// TIA Portal V19 export
FUNCTION "APP_UPDATE STEP NO. UHT" : Void   // FC30, STL
TITLE = Step update to OP25
{ S7_Optimized_Access := 'TRUE' }
AUTHOR : JOM
FAMILY : APP
NAME : STEP_UPD
// Main Update:       1 = Start                     7 = Stop production     
//                    2 = Presterilizing            8 = Recirculation water
//                    3 = Stop presteril            9 = Stop recirculation water
//                    4 = Cip                      10 = Aseptic cip
//                    5 = Stop cip                 11 = Stop aseptic cip
//                    6 = Production               12 = Total stop
//                    13 = CIP FILLER
// 
// Step Update:     101 = Standby             102-110 = Start     
//              111-120 = Presterilizing      121-130 = Stop presteril
//              131-154 = Cip                 155-160 = Stop Cip
//              161-170 = Production          171-180 = Stop production            
//              181-190 = Total stop              200 = Error step tank
//              201-250 = CIP FILLER
// ****** REVISION HISTORY :
// 
// VERSION DATE         BY    DESCRIPTION
// --------------------------------------------------------------------------
// 00.00   25/9 1997   OPA   ORIGINAL FUNCTION BLOCK
//       
// 00.01   11/2 1998   OPA   STOP CIP ADDED
//  
// SOFTWARE SIMULATED IN OFFICE *******DATE*********
// stored: AutoNumber false
BEGIN

NETWORK
TITLE = 
      CLR;
      A     "Tag_74";
      BEC;

      AN    "ViewUHT_TANK_OP25";
      JC    TANK;


NETWORK
TITLE = 
      A     "S0 FILLER";
      ON    "ViewUHT_TANK_OP25";
      JC    FIL0;
      L     0;
      T     "OP25 TANK".TaStepUpdating;
      T     "OP25 TANK".TaMainUpdating;


FIL0: A     "S0 FILLER";  //"S0 CIP TANK"
      AN    "S16 FILLER";  //"S16 CIP TANK"
      JCN   FIL1;

      CALL  "STD_UPDATE_STEP_OP25"
      ( START      := "S0 FILLER",
        FLAG_WORD  := "Tag_18",
        OFFSET     := 200,
        MAX        := 16,
        MAIN_NO    := 13,
        OLD_STATUS := "StepOldStatus",
        COUNT      := "OP25 TANK".TaStepUpdating,
        MAIN       := "OP25 TANK".TaMainUpdating
      );
      BEU;

FIL1: A     "S16 FILLER";  //"S0 CIP TANK"
      AN    "S32 FILLER";  //"S16 CIP TANK"
      JCN   FIL3;



      A     "S15 FILLER";  // THE FC-STANDARD BLOCK CANNOT
      AN    "S16 FILLER";  // DEAL WITH MORE THAN 16 STEP (=WORD)
      JCN   FIL2;  // IN EACH FUNCTION. ALL BITS IN MW118
      L     13;  // ARE HIGH AND NO BIT IS SET IN MW120.
      T     "OP25 TANK".TaMainUpdating;  // FOR THE SPECIAL CASE: WAITING FOR
      L     216;  // FOR M120.0 TO BE HIGH, THEN
      T     "OP25 TANK".TaStepUpdating;  // TRANSFER VALUES MANUAL.

FIL2: CALL  "STD_UPDATE_STEP_OP25"
      ( START      := "S16 FILLER",
        FLAG_WORD  := "Tag_19",
        OFFSET     := 216,
        MAX        := 16,
        MAIN_NO    := 13,
        OLD_STATUS := "StepOldStatus",
        COUNT      := "OP25 TANK".TaStepUpdating,
        MAIN       := "OP25 TANK".TaMainUpdating
      );  //UPDATE REMAINING STEPS IN CIP
      BEU;
//
FIL3: A     "S31 FILLER";  // THE FC-STANDARD BLOCK CANNOT
      AN    "S32 FILLER";  // DEAL WITH MORE THAN 16 STEP (=WORD)
      JCN   FIL4;  // IN EACH FUNCTION. ALL BITS IN MW118
      L     13;  // ARE HIGH AND NO BIT IS SET IN MW120.
      T     "OP25 TANK".TaMainUpdating;  // FOR THE SPECIAL CASE: WAITING FOR
      L     232;  // FOR M120.0 TO BE HIGH, THEN
      T     "OP25 TANK".TaStepUpdating;  // TRANSFER VALUES MANUAL.



FIL4: CALL  "STD_UPDATE_STEP_OP25"
      ( START      := "S32 FILLER",
        FLAG_WORD  := "Tag_20",
        OFFSET     := 232,
        MAX        := 14,
        MAIN_NO    := 13,
        OLD_STATUS := "StepOldStatus",
        COUNT      := "OP25 TANK".TaStepUpdating,
        MAIN       := "OP25 TANK".TaMainUpdating
      );  //
      NOP   0;
      BEU;


NETWORK
TITLE = UPDATE FUNCTION AND STEP IN PRESTERILIZING
// Presterilizing  111-120
TANK: AN    "TANK AUTO";
      L     0;
      T     "OP25 TANK".TaMainUpdating;
      T     "OP25 TANK".TaStepUpdating;
      BEC;

      CALL  "STD_UPDATE_STEP_OP25"
      ( START      := "S0 PRESTERILIZING",
        FLAG_WORD  := "Tag_21",
        OFFSET     := 110,
        MAX        := 8,
        MAIN_NO    := 2,
        OLD_STATUS := "StepOldStatus",
        COUNT      := "OP25 TANK".TaStepUpdating,
        MAIN       := "OP25 TANK".TaMainUpdating
      );  //


NETWORK
TITLE = UPDATE FUNCTION AND STEP IN STOP PRESTERILIZING
// Stop presterilizing   121-130
      CALL  "STD_UPDATE_STEP_OP25"
      ( START      := "S0 STOP PRESTE. TANK",
        FLAG_WORD  := "Tag_22",
        OFFSET     := 120,
        MAX        := 4,
        MAIN_NO    := 3,
        OLD_STATUS := "StepOldStatus",
        COUNT      := "OP25 TANK".TaStepUpdating,
        MAIN       := "OP25 TANK".TaMainUpdating
      );  //


NETWORK
TITLE = UPDATE FUNCTION AND STEP IN CIP
// Cip   131-154
      A     "S0 CIP TANK";
      AN    "S16 CIP TANK";
      JCN   CIP1;

      CALL  "STD_UPDATE_STEP_OP25"
      ( START      := "S0 CIP TANK",
        FLAG_WORD  := "Tag_23",
        OFFSET     := 130,
        MAX        := 16,
        MAIN_NO    := 4,
        OLD_STATUS := "StepOldStatus",
        COUNT      := "OP25 TANK".TaStepUpdating,
        MAIN       := "OP25 TANK".TaMainUpdating
      );

CIP1: A     "S15 CIP TANK";  // THE FC-STANDARD BLOCK CANNOT
      AN    "S16 CIP TANK";  // DEAL WITH MORE THAN 16 STEP (=WORD)
      JCN   CIP2;  // IN EACH FUNCTION. ALL BITS IN MW118
      L     4;  // ARE HIGH AND NO BIT IS SET IN MW120.
      T     "OP25 TANK".TaMainUpdating;  // FOR THE SPECIAL CASE: WAITING FOR
      L     146;  // FOR M120.0 TO BE HIGH, THEN
      T     "OP25 TANK".TaStepUpdating;  // TRANSFER VALUES MANUAL.

CIP2: CALL  "STD_UPDATE_STEP_OP25"
      ( START      := "S16 CIP TANK",
        FLAG_WORD  := "Tag_24",
        OFFSET     := 146,
        MAX        := 5,
        MAIN_NO    := 4,
        OLD_STATUS := "StepOldStatus",
        COUNT      := "OP25 TANK".TaStepUpdating,
        MAIN       := "OP25 TANK".TaMainUpdating
      );  //UPDATE REMAINING STEPS IN CIP
//

NETWORK
TITLE = UPDATE FUNCTION AND STEP IN STOP CIP
// CIP   155-160
      CALL  "STD_UPDATE_STEP_OP25"
      ( START      := "S0 STOP CIP TANK",
        FLAG_WORD  := "Tag_25",
        OFFSET     := 154,
        MAX        := 4,
        MAIN_NO    := 5,
        OLD_STATUS := "StepOldStatus",
        COUNT      := "OP25 TANK".TaStepUpdating,
        MAIN       := "OP25 TANK".TaMainUpdating
      );  //
//

NETWORK
TITLE = UPDATE FUNCTION AND STEP IN PRODUCTION
// Production   161-170
      CALL  "STD_UPDATE_STEP_OP25"
      ( START      := "S0 PRODUCTION TANK",
        FLAG_WORD  := "Tag_26",
        OFFSET     := 160,
        MAX        := 3,
        MAIN_NO    := 6,
        OLD_STATUS := "StepOldStatus",
        COUNT      := "OP25 TANK".TaStepUpdating,
        MAIN       := "OP25 TANK".TaMainUpdating
      );  //
//

NETWORK
TITLE = UPDATE FUNCTION AND STEP IN STOP PRODUCTION
// Stop production   171-180
      CALL  "STD_UPDATE_STEP_OP25"
      ( START      := "S0 STOP PRODUCTION TANK",
        FLAG_WORD  := "Tag_27",
        OFFSET     := 170,
        MAX        := 3,
        MAIN_NO    := 7,
        OLD_STATUS := "StepOldStatus",
        COUNT      := "OP25 TANK".TaStepUpdating,
        MAIN       := "OP25 TANK".TaMainUpdating
      );  //
//

NETWORK
TITLE = UPDATE FUNCTION AND STEP IN TOTAL STOP TANK
// TOTAL STOP TANK   181-190
      CALL  "STD_UPDATE_STEP_OP25"
      ( START      := "S0 TOTAL STOP TANK",
        FLAG_WORD  := "Tag_28",
        OFFSET     := 180,
        MAX        := 3,
        MAIN_NO    := 12,
        OLD_STATUS := "StepOldStatus",
        COUNT      := "OP25 TANK".TaStepUpdating,
        MAIN       := "OP25 TANK".TaMainUpdating
      );  //
//
END_FUNCTION
